Fanuc KAREL source: kb00116.KL

-- PROVISIONAL review KL for V1013-1; original PC SHA256 95841b72f029f8bcb7715fc70c81621787f2997e9ee530a795ca24836d7c179b
-- Incomplete behavior may be omitted. Consult companion uncertainty JSON. Do not deploy.
PROGRAM KB00116
%NOLOCKGROUP
VAR
  P1 : REAL
  RESULT : REAL
BEGIN
  -- UNRESOLVED_PC offsets 5-16; opcodes 2E,23
  -- UNRESOLVED_PC offsets 21-36; opcodes 27,22,76,23
  -- UNRESOLVED_PC offsets 41-45; opcodes 7F
END KB00116
